PROGRAM valve_analog_control
VAR PERSISTENT
	// Example Analog Valve Function Block
	av_3148: valve_analog;
END_VAR

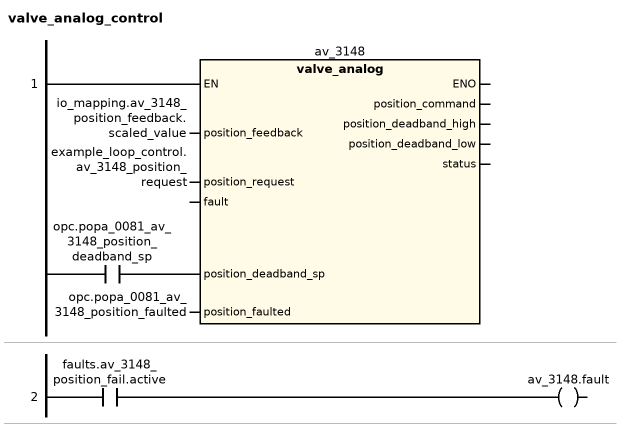
// NETWORK 1
av_3148(
    position_feedback := io_mapping.av_3148_position_feedback.scaled_value,
    position_request := example_loop_control.av_3148_position_request,
    position_deadband_sp := opc.popa_0081_av_3148_position_deadband_sp,
    position_faulted := opc.popa_0081_av_3148_position_faulted); // valve_analog

// NETWORK 2
av_3148.fault := faults.av_3148_position_fail.active;

END_PROGRAM

(* stored: Version 1.1.0.1, ProductVersion 3.1.4024.12
   POU valve_analog_control: Id {54a66418-c0f3-4155-b95b-fc459b2a3fbb}, SpecialFunc None *)
